(* IEC 61131-3 sources: Std_PalletMover/Class/ManualControl, 1 file *)

(* ---- ManualControl.st ---- *)
(*!
<Class
	Name               = "ManualControl"
	Revision           = "0.0"
	RealtimeTask       = "false"
	CyclicTask         = "false"
	BackgroundTask     = "false"
	Sigmatek           = "false"
	OSInterface        = "false"
	HighPriority       = "false"
	Automatic          = "false"
	UpdateMode         = "Prescan"
	SharedCommandTable = "true"
	Objectsize         = "(720,120)">
	<Channels>
		<Server Name="AgvManualControl" Visualized="false" Initialize="true" WriteProtected="true" Retentive="false"/>
	</Channels>
	<Network Name="ManualControl">
		<!-- List of Components in this network -->
		<Components>
			<Object
				Name       = "_base"
				Class      = "WewoBase"
				Position   = "(218,120)"
				Visualized = "false">
				<Channels>
					<Server Name="m_Id"/>
					<Server Name="m_p_Name"/>
					<Server Name="o_ErrorWarningStatus"/>
					<Server Name="ObjectStatus"/>
					<Server Name="ToObject"/>
					<Client Name="c_Group"/>
					<Client Name="op_LogData"/>
					<Client Name="toOsLibTaskObjControl"/>
				</Channels>
			</Object>
		</Components>
		<Comments>
		</Comments>
		<!-- List of Connections in this network -->
		<Connections>
			<Connection Source="this.ToObject" Destination="_base.ToObject" Vertices="(856,210),(684,210),"/>
		</Connections>
		<!-- Headerfiles -->
		<Options>
		</Options>
	</Network>
</Class>
*)
#pragma using WewoBase

ManualControl : CLASS
: WewoBase
  //Servers:
	AgvManualControl 	: SvrCh_gt_AgvManual;
  //Clients:
  //Variables:
  //Functions:

	FUNCTION GLOBAL MainAutoControl;
  //Tables:
	FUNCTION @STD
		VAR_OUTPUT
			ret_code	: CONFSTATES;
		END_VAR;
	FUNCTION GLOBAL TAB @CT_;
END_CLASS;

FUNCTION GLOBAL ManualControl::MainAutoControl

    // wait for Program from mes

    // Start Program

    // init step

    // Exec step

        // wait ready

END_FUNCTION
